ABB RobotStudio station: Lab-1.rsstnx

Station Lab-1 (saved by RobotStudio 24.3.10885.0)
Controller IRB120_3_58
  mechanical unit ROB_1: IRB120T_3_58__01, 6 joints, base frame (0, 0, 0) mm
Layout (positions relative to the parent item):
  - IRB120T_3_58__01 [mechanism, from %ABB.RobotStudio.Models.IRB120%\IRB120T_3_58_G_01.rslib] at (0, 0, 0) mm; joint values [0, 0, 0, 0, 0.5236, 0] (rad or m)
